Omron Sysmac Studio project Husillo_F3 (Sysmac Studio 1.23.0.14, StandardProject)

# Controller new_Controller_0: NX1P2-1040DT1 version 1.18
Task PrimaryTask (priority 4, period or condition 2000): Programa0

VAR_GLOBAL
    PP : BOOL;  (* Pulsador Paro; at BuiltInIO://cpu/#0/Input_Bit_00 *)
    PM : BOOL;  (* Pulsador Marcha; at BuiltInIO://cpu/#0/Input_Bit_01 *)
    PR : BOOL;  (* Pulsador Reset; at BuiltInIO://cpu/#0/Input_Bit_02 *)
    FCI : BOOL;  (* Final Carrera Izquierda; at BuiltInIO://cpu/#0/Input_Bit_03 *)
    FCD : BOOL;  (* Final Carrera Derecha; at BuiltInIO://cpu/#0/Input_Bit_04 *)
    V1 : BOOL;  (* Motor Derecha; at BuiltInIO://cpu/#0/Output_Bit_00 *)
    V2 : BOOL;  (* Motor Izquierda; at BuiltInIO://cpu/#0/Output_Bit_01 *)
    PP_HMI AT %W0.00 : BOOL;  (* Pulsador Paro HMI; published *)
    PM_HMI AT %W0.01 : BOOL;  (* Pulsador Marcha HMI; published *)
    PR_HMI AT %W0.02 : BOOL;  (* Pulsador Reset HMI; published *)
END_VAR
VAR_GLOBAL RETAIN
    STATE AT %D10 : DINT;  (* published *)
END_VAR

PROGRAM Programa0
VAR
    Et0 : BOOL;  (* Etapa 0 *)
    Et1 : BOOL;  (* Etapa 1 *)
    Et2 : BOOL;  (* Etapa 2 *)
    Et3 : BOOL;  (* Etapa 3 *)
    Et4 : BOOL;  (* Etapa 4 *)
    Et10 : BOOL;  (* Etapa 10 *)
    Et11 : BOOL;  (* Etapa 11 *)
    Et12 : BOOL;  (* Etapa 12 *)
    PM_V : BOOL;  (* Pulsador Marcha *)
    PP_V : BOOL;  (* Pulsador Paro *)
    PR_V : BOOL;  (* Pulsador Reset *)
    C1 : CTU;
    T1 : TON;
    Iterations : INT;
END_VAR
VAR_EXTERNAL
    FCD : BOOL;
    PM : BOOL;
    FCI : BOOL;
    PP : BOOL;
    PR : BOOL;
    V1 : BOOL;
    V2 : BOOL;
    PP_HMI : BOOL;
    PR_HMI : BOOL;
    STATE : DINT;
END_VAR
VAR
    _e1 : R_TRIG;
END_VAR

(* Section Main: ladder, written here as Structured Text *)

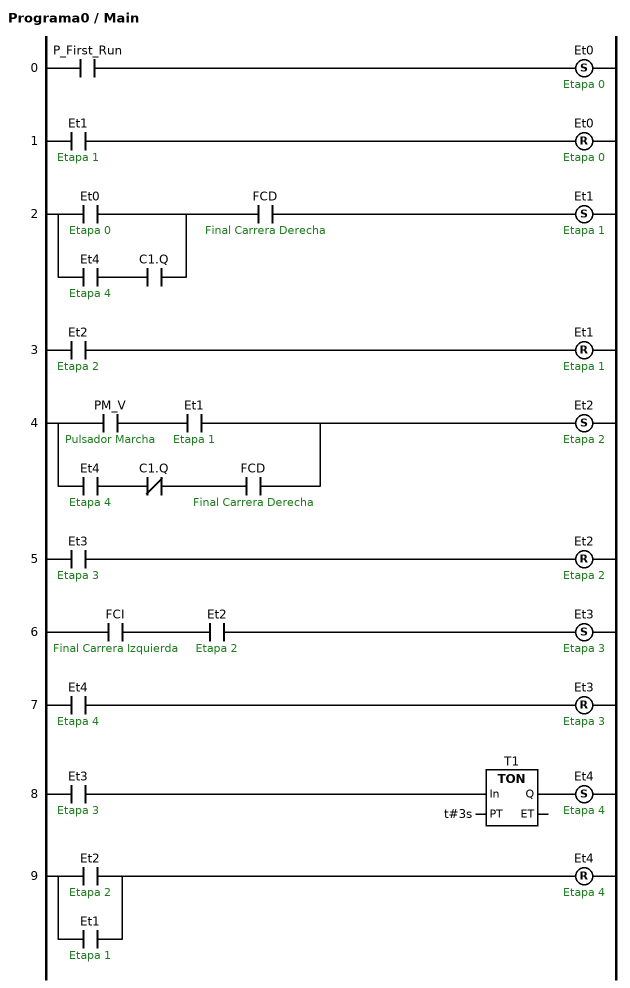
(* Rung 0 *)
IF P_First_Run THEN Et0 := TRUE; END_IF;
(* Rung 1 *)
IF Et1 THEN Et0 := FALSE; END_IF;
(* Rung 2 *)
IF (Et0 OR (Et4 AND C1.Q)) AND FCD THEN Et1 := TRUE; END_IF;
(* Rung 3 *)
IF Et2 THEN Et1 := FALSE; END_IF;
(* Rung 4 *)
IF (PM_V AND Et1) OR (Et4 AND NOT C1.Q AND FCD) THEN Et2 := TRUE; END_IF;
(* Rung 5 *)
IF Et3 THEN Et2 := FALSE; END_IF;
(* Rung 6 *)
IF FCI AND Et2 THEN Et3 := TRUE; END_IF;
(* Rung 7 *)
IF Et4 THEN Et3 := FALSE; END_IF;
(* Rung 8 *)
T1(In := Et3, PT := t#3s);
IF T1.Q THEN Et4 := TRUE; END_IF;
(* Rung 9 *)
IF Et2 OR Et1 THEN Et4 := FALSE; END_IF;

(* Section Reset: ladder, written here as Structured Text *)

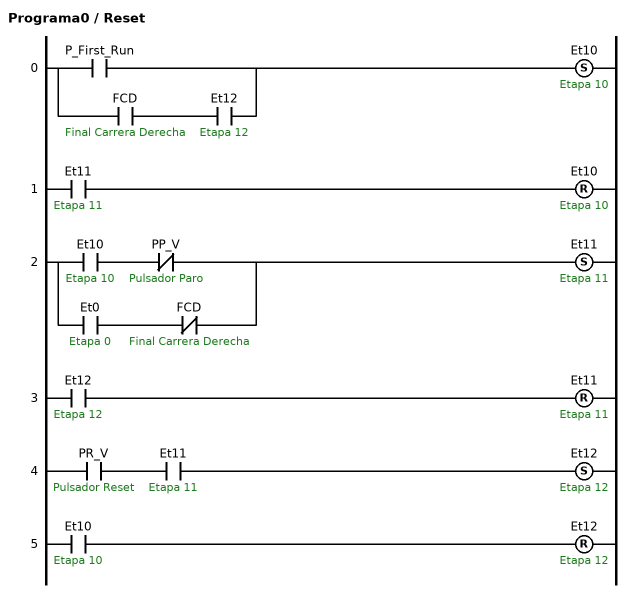
(* Rung 0 *)
IF P_First_Run OR (FCD AND Et12) THEN Et10 := TRUE; END_IF;
(* Rung 1 *)
IF Et11 THEN Et10 := FALSE; END_IF;
(* Rung 2 *)
IF (Et10 AND NOT PP_V) OR (Et0 AND NOT FCD) THEN Et11 := TRUE; END_IF;
(* Rung 3 *)
IF Et12 THEN Et11 := FALSE; END_IF;
(* Rung 4 *)
IF PR_V AND Et11 THEN Et12 := TRUE; END_IF;
(* Rung 5 *)
IF Et10 THEN Et12 := FALSE; END_IF;

(* Section Outputs: ladder, written here as Structured Text *)

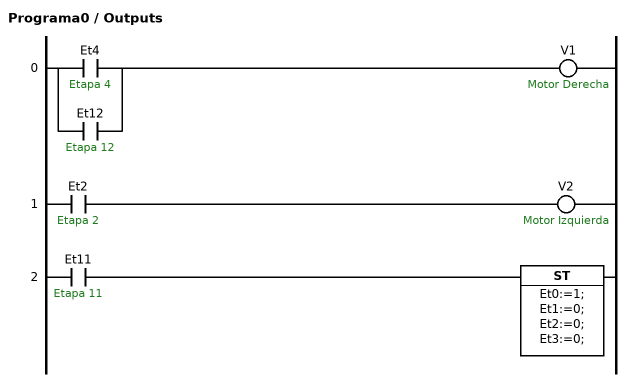
(* Rung 0 *)
V1 := Et4 OR Et12;
(* Rung 1 *)
V2 := Et2;
(* Rung 2 *)
IF Et11 THEN
    Et0:=1;
    Et1:=0;
    Et2:=0;
    Et3:=0;
END_IF;

(* Section IO_Merge: ladder, written here as Structured Text *)

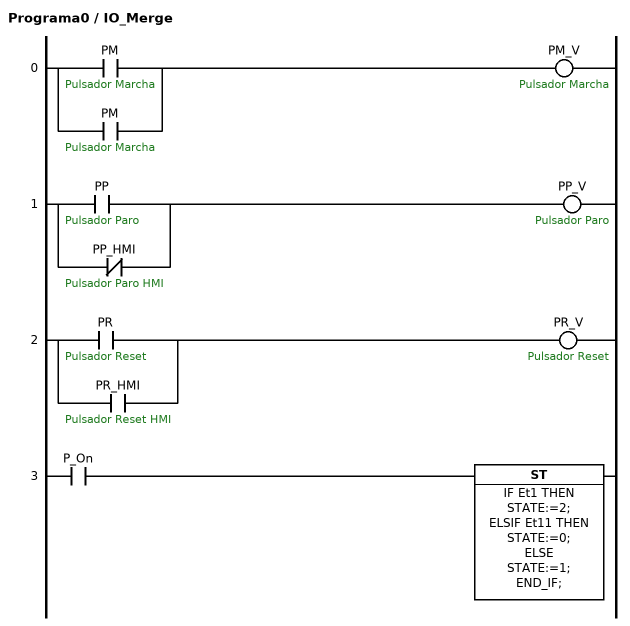
(* Rung 0 *)
PM_V := PM OR PM;
(* Rung 1 *)
PP_V := PP OR NOT PP_HMI;
(* Rung 2 *)
PR_V := PR OR PR_HMI;
(* Rung 3 *)
IF P_On THEN
    IF Et1 THEN
        STATE:=2;
    ELSIF Et11 THEN
        STATE:=0;
    ELSE
        STATE:=1;
    END_IF;
END_IF;

(* Section Counter: ladder, written here as Structured Text *)

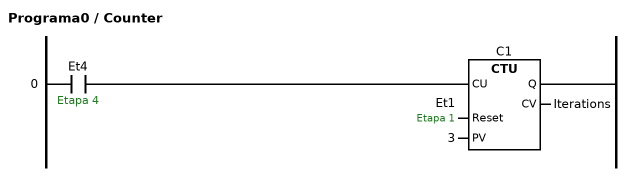
(* Rung 0 *)
_e1(CLK := Et4);
C1(CU := _e1.Q, Reset := Et1, PV := 3, CV => Iterations);
END_PROGRAM